// TIA Portal V20 export
TYPE "LKinCtrl_typePointCoordinates"
   STRUCT
      cartesianPosition : "LKinCtrl_typeCartesianPosition";   // cartesian position
      coordSystem : DInt := 0;   // 0: WCS; 1: OCS[1]; 2: OCS[2]; 3: OCS[3]; 100: MCS
   END_STRUCT;
END_TYPE
